// TwinCAT 3 PLC project HMI_Hemo
// ProgramVersion: 3.1.4024.0
// libraries:
//   Tc2_Standard, * (Beckhoff Automation GmbH)
//   Tc2_System, * (Beckhoff Automation GmbH)
//   Tc3_Module, * (Beckhoff Automation GmbH)
//   VisuDialogs, * (System)
//   VisuSymbols,3.5.10.0,System
// project tree:
//   / GlobalTextList.TcGTLO, PlcTask.TcTTO, Visualization Manager.TcVMO (not stored), VISU_TASK.TcTTO
//   GVLs/ GVL.TcGVL
//   POUs/ MAIN.TcPOU
//   VISUs/ Main_Screen.TcVIS, Screen_1.TcVIS, Screen_Maintenance.TcVIS, Screen_1_Sub_1.TcVIS, Screen_1_Sub_2.TcVIS, Screen_1_Sub_3.TcVIS, Screen_1_Sub_4.TcVIS, Screen_3.TcVIS, Screen_3_Sub_1.TcVIS, Screen_2_Sub_1.TcVIS, Screen_2.TcVIS, Screen_2_Sub_2.TcVIS, Screen_2_Sub_7.TcVIS, Screen_2_Sub_6.TcVIS, Screen_2_Sub_3.TcVIS, Screen_2_Sub_4.TcVIS, Screen_2_Sub_5.TcVIS, Screen_Prep.TcVIS, Screen_Rinse.TcVIS, Screen_Dialys.TcVIS
// real-time tasks:
//   TASK PlcTask: cycle T#10ms, priority 20, ADS port 350
//   TASK VISU_TASK: cycle T#200000us, priority 30, ADS port 351

CONFIGURATION HMI_Hemo
    RESOURCE PLC ON TwinCAT3
        TASK PlcTask(INTERVAL := T#10ms, PRIORITY := 20);
        TASK VISU_TASK(INTERVAL := T#200000us, PRIORITY := 30);
        PROGRAM MAIN WITH PlcTask : MAIN;
        PROGRAM VisuElems_Visu_Prg WITH VISU_TASK : VisuElems.Visu_Prg;
    END_RESOURCE
END_CONFIGURATION

// ---- GVLs/GVL.TcGVL
{attribute 'qualified_only'}
VAR_GLOBAL
	
	// HMI State ON/OFF
	HMI_State_ON_OFF				: BOOL;
	
	// HMI Variable Global Heading
	HMI_Heading						: ARRAY[0..2] OF INT;
	
	// HMI Variable Prep
	HMI_Prep_Name_Display			: ARRAY[0..7] OF STRING;
	HMI_Prep_Name_Input				: ARRAY[0..3] OF STRING;
	HMI_Prep_Name_IO				: ARRAY[0..3] OF STRING;
	
	HMI_Prep_Display_Var			: ARRAY[0..7] OF INT;
	HMI_Prep_Input_Var				: ARRAY[0..3] OF INT;
	HMI_Prep_IO_Var					: ARRAY[0..3] OF BOOL;
	
	// HMI Variable Rinse
	HMI_Rinse_Name_Display			: ARRAY[0..7] OF STRING;
	HMI_Rinse_Name_Input				: ARRAY[0..3] OF STRING;
	HMI_Rinse_Name_IO				: ARRAY[0..3] OF STRING;
	
	HMI_Rinse_Display_Var			: ARRAY[0..7] OF INT;
	HMI_Rinse_Input_Var				: ARRAY[0..3] OF INT;
	HMI_Rinse_IO_Var				: ARRAY[0..3] OF BOOL;
	
	// HMI Variable Dialys
	HMI_Dialys_Name_Display			: ARRAY[0..7] OF STRING;
	HMI_Dialys_Name_Input			: ARRAY[0..3] OF STRING;
	HMI_Dialys_Name_IO				: ARRAY[0..3] OF STRING;
	
	HMI_Dialys_Display_Var			: ARRAY[0..7] OF INT;
	HMI_Dialys_Input_Var			: ARRAY[0..3] OF INT;
	HMI_Dialys_IO_Var				: ARRAY[0..3] OF BOOL;
	
	// HMI Variable Global Declaration
	
	HMI_Button_Valve				: ARRAY[0..31] OF BOOL;
	HMI_Display_Int					: ARRAY[0..31] OF INT;
	HMI_Display_Lamp				: ARRAY[0..31] OF BOOL;

	HMI_Motor_Peristaltik_Input 	: INT;
	HMI_Motor_Peristaltik_Real		: INT;
	
	HMI_Motor_DAC_1_Input			: INT;
	HMI_Motor_DAC_1_Real			: INT;
	
	HMI_Motor_DAC_2_Input			: INT;
	HMI_Motor_DAC_2_Real			: INT;
	
	HMI_Motor_Pump_1_Input			: INT;
	HMI_Motor_Pump_1_Real			: INT;
	
	HMI_Motor_Pump_2_Input			: INT;
	HMI_Motor_Pump_2_Real			: INT;
	
	HMI_Motor_Pump_3_Input			: INT;
	HMI_Motor_Pump_3_Real			: INT;
	
	HMI_Motor_Stepper_Input			: INT;
	HMI_Motor_Stepper_Real			: INT;
	HMI_Motor_Stepper_Injec_Stat	: BOOL;
	HMI_Motor_Stepper_Zero_Pos		: BOOL;
	
	HMI_Number_Display				: ARRAY[0..31] OF INT;
	
	//HMI Variable for Maintenance
	
	HMI_Maintenance_H				: BOOL;	
	HMI_Maintenance_P1				: BOOL;	
	HMI_Maintenance_P2				: BOOL;	
	HMI_Maintenance_P3				: BOOL;	
	HMI_Maintenance_P4				: BOOL;	
	
	HMI_Maintenance_V1				: BOOL;	
	HMI_Maintenance_V4				: BOOL;	
	HMI_Maintenance_V5A				: BOOL;	
	HMI_Maintenance_V5B				: BOOL;	
	HMI_Maintenance_V6A				: BOOL;	
	HMI_Maintenance_V6B				: BOOL;	
	HMI_Maintenance_V7A				: BOOL;	
	HMI_Maintenance_V7B				: BOOL;	
	HMI_Maintenance_V8A				: BOOL;	
	HMI_Maintenance_V8B				: BOOL;	
	HMI_Maintenance_V9A				: BOOL;	
	HMI_Maintenance_V9B				: BOOL;

	HMI_Maintenance_V10				: BOOL; 
	HMI_Maintenance_V11				: BOOL;
	HMI_Maintenance_V12				: BOOL;
	HMI_Maintenance_V17				: BOOL;
	HMI_Maintenance_V19				: BOOL;
	HMI_Maintenance_V21				: BOOL;
	HMI_Maintenance_V24				: BOOL;
	HMI_Maintenance_V27				: BOOL;
	HMI_Maintenance_V28				: BOOL;
	HMI_Maintenance_V29				: BOOL;
	HMI_Maintenance_V30				: BOOL;
	HMI_Maintenance_V31				: BOOL;
	
	HMI_Maintenance_V33				: BOOL;	
	HMI_Maintenance_V34				: BOOL;
	HMI_Maintenance_V35				: BOOL;
	HMI_Maintenance_V43				: BOOL;
	HMI_Maintenance_V45				: BOOL;
	HMI_Maintenance_V46				: BOOL;
	HMI_Maintenance_V55				: BOOL;
	HMI_Maintenance_V56				: BOOL;
	HMI_Maintenance_V57				: BOOL;
	
	
	
END_VAR

// ---- POUs/MAIN.TcPOU
PROGRAM MAIN
VAR	

END_VAR

// GVL Variable For Prep
GVL.HMI_Prep_Name_Display[0] := 'Test';
GVL.HMI_Prep_Name_Display[1] := 'Test';
GVL.HMI_Prep_Name_Display[2] := 'Test';
GVL.HMI_Prep_Name_Display[3] := 'Test';
GVL.HMI_Prep_Name_Display[4] := 'Test';
GVL.HMI_Prep_Name_Display[5] := 'Test';
GVL.HMI_Prep_Name_Display[6] := 'Test';
GVL.HMI_Prep_Name_Display[7] := 'Test';

GVL.HMI_Prep_Name_Input[0] := 'Test';
GVL.HMI_Prep_Name_Input[1] := 'Test';
GVL.HMI_Prep_Name_Input[2] := 'Test';
GVL.HMI_Prep_Name_Input[3] := 'Test';

GVL.HMI_Prep_Name_IO[0] := 'Test';
GVL.HMI_Prep_Name_IO[1] := 'Test';
GVL.HMI_Prep_Name_IO[2] := 'Test';
GVL.HMI_Prep_Name_IO[3] := 'Test';

END_PROGRAM

// ---- GlobalTextList.TcGTLO
TEXTLIST GlobalTextList
  52 = ' Val 10: %i'
  420 = ' Val 11: %i'
  658 = ' Val 12: %i'
  696 = ' Val 13: %i'
  313 = ' Val 14: %i'
  1050 = ' Val 15: %i'
  862 = ' Val 16: %i'
  715 = ' Val 17: %i'
  463 = ' Val 18: %i'
  761 = ' Val 19: %i'
  366 = ' Val 1: %i'
  822 = ' Val 20: %i'
  648 = ' Val 21: %i'
  318 = ' Val 22: %i'
  1131 = ' Val 23: %i'
  134 = ' Val 24: %i'
  689 = ' Val 25: %i'
  59 = ' Val 26: %i'
  29 = ' Val 27: %i'
  476 = ' Val 28: %i'
  911 = ' Val 29: %i'
  161 = ' Val 2: %i'
  193 = ' Val 30: %i'
  656 = ' Val 31: %i'
  579 = ' Val 32: %i'
  849 = ' Val 3: %i'
  159 = ' Val 4: %i'
  380 = ' Val 5: %i'
  207 = ' Val 6: %i'
  261 = ' Val 7: %i'
  42 = ' Val 8: %i'
  58 = ' Val 9: %i'
  1018 = '%i'
  1046 = '%s'
  1856 = 'Diagram'
  61 = 'DIALYS'
  1024 = 'Dialys Mode'
  1006 = 'Digital Input'
  1260 = 'Display Variable'
  28 = 'dsfads'
  1374 = 'H'
  608 = 'Injection Status'
  112 = 'Input 1'
  162 = 'Input 10'
  462 = 'Input 11'
  577 = 'Input 12'
  944 = 'Input 13'
  742 = 'Input 14'
  680 = 'Input 15'
  475 = 'Input 16'
  273 = 'Input 17'
  127 = 'Input 18'
  208 = 'Input 19'
  816 = 'Input 2'
  306 = 'Input 20'
  515 = 'Input 21'
  972 = 'Input 22'
  70 = 'Input 23'
  242 = 'Input 24'
  779 = 'Input 25'
  714 = 'Input 26'
  84 = 'Input 27'
  53 = 'Input 28'
  228 = 'Input 29'
  471 = 'Input 3'
  343 = 'Input 30'
  745 = 'Input 31'
  808 = 'Input 32'
  566 = 'Input 4'
  775 = 'Input 5'
  874 = 'Input 6'
  599 = 'Input 7'
  359 = 'Input 8'
  440 = 'Input 9'
  1650 = 'Input Output'
  543 = 'Input Variable'
  1242 = 'Kecepatan Real'
  393 = 'Konfigurasi Input Output'
  931 = 'Konfigurasi Motor'
  633 = 'Lamp 1'
  1869 = 'Maintanance'
  1561 = 'Maintenance'
  544 = 'MAINTENANCE'
  45 = 'Mesin Hemodialisis'
  56 = 'Motor'
  131 = 'Motor DAC 1'
  1109 = 'Motor DAC 2'
  194 = 'Motor Peristaltik'
  744 = 'Motor Pump 1'
  1236 = 'Motor Pump 2'
  304 = 'Motor Pump 3'
  1002 = 'Motor Stepper'
  1079 = 'Num Display 1'
  311 = 'Num Display 2'
  1150 = 'Number Display 1'
  1017 = 'Number Display 2'
  1036 = 'off'
  1043 = 'OFF'
  1929 = 'ON/OFF'
  817 = 'P1'
  60 = 'P2'
  815 = 'P2H'
  649 = 'P3'
  930 = 'P4'
  1144 = 'PREP'
  367 = 'Prep Mode'
  1822 = 'Preparation'
  1625 = 'RINSE'
  1635 = 'Rinse Mode'
  982 = 'Setpoint Kecepatan'
  1174 = 'Tombol Valve'
  678 = 'V1'
  1333 = 'V10'
  617 = 'V11'
  1375 = 'V12'
  1051 = 'V17'
  912 = 'V19'
  1674 = 'V21'
  618 = 'V24'
  542 = 'v27'
  4 = 'V27'
  846 = 'V28'
  922 = 'V29'
  1189 = 'V30'
  510 = 'V31'
  1373 = 'V33'
  1492 = 'V34'
  1774 = 'V35'
  1487 = 'V4'
  593 = 'V43'
  49 = 'V45'
  191 = 'v46'
  101 = 'V46'
  1268 = 'V55'
  1183 = 'V56'
  108 = 'V57'
  66 = 'V5A'
  182 = 'V5a'
  1304 = 'V5b'
  436 = 'V6a'
  1520 = 'V6b'
  468 = 'V7a'
  1310 = 'V7b'
  971 = 'V8a'
  759 = 'V8b'
  200 = 'V9a'
  1329 = 'V9b'
  691 = 'Val 10: %i'
  270 = 'Val 11: %i'
  100 = 'Val 12: %i'
  408 = 'Val 13: %i'
  771 = 'Val 14: %i'
  692 = 'Val 15: %i'
  807 = 'Val 16: %i'
  281 = 'Val 17: %i'
  948 = 'Val 18: %i'
  457 = 'Val 19: %i'
  54 = 'Val 1: %i'
  426 = 'Val 20: %i'
  79 = 'Val 21: %i'
  128 = 'Val 22: %i'
  929 = 'Val 23: %i'
  902 = 'Val 24: %i'
  32 = 'Val 25: %i'
  238 = 'Val 26: %i'
  549 = 'Val 27: %i'
  379 = 'Val 28: %i'
  418 = 'Val 29: %i'
  917 = 'Val 2: %i'
  886 = 'Val 30: %i'
  629 = 'Val 31: %i'
  155 = 'Val 32: %i'
  981 = 'Val 3: %i'
  877 = 'Val 4: %i'
  26 = 'Val 5: %i'
  333 = 'Val 6: %i'
  612 = 'Val 7: %i'
  31 = 'Val 8: %i'
  220 = 'Val 9: %i'
  55 = 'Valve 1'
  964 = 'Valve 10'
  3 = 'Valve 11'
  265 = 'Valve 12'
  952 = 'Valve 13'
  357 = 'Valve 14'
  65 = 'Valve 15'
  664 = 'Valve 16'
  121 = 'Valve 17'
  578 = 'Valve 18'
  589 = 'Valve 19'
  391 = 'Valve 2'
  2 = 'Valve 20'
  954 = 'Valve 21'
  107 = 'Valve 22'
  174 = 'Valve 23'
  934 = 'Valve 24'
  67 = 'Valve 25'
  734 = 'Valve 26'
  354 = 'Valve 27'
  968 = 'Valve 28'
  879 = 'Valve 29'
  502 = 'Valve 3'
  137 = 'Valve 30'
  340 = 'Valve 31'
  348 = 'Valve 32'
  733 = 'Valve 4'
  467 = 'Valve 5'
  227 = 'Valve 6'
  22 = 'Valve 7'
  977 = 'Valve 8'
  737 = 'Valve 9'
  465 = 'Variable Input Output'
  1258 = 'Zero Pos Status'
  464 = 'Zero Position Status'
END_TEXTLIST

// ---- VISUs/Main_Screen.TcVIS
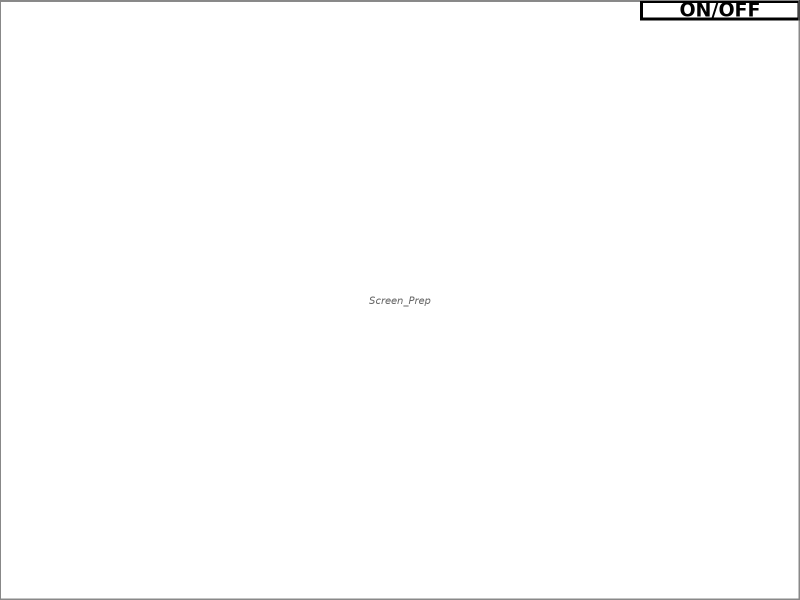
VISUALIZATION Main_Screen  // 800x600
    TabControl (0,1 800x599), frame switch variable: GVL.HMI_Heading[0]
        shows Screen_Prep()
        shows Screen_Rinse()
        shows Screen_Dialys()
        shows Screen_Maintenance()
        [0]: TabTitle=Prep Mode
        [1]: TabTitle=Rinse Mode
        [2]: TabTitle=Dialys Mode
        [3]: TabTitle=Maintenance
    Rectangle (640,0 160x20), "ON/OFF", colour toggle: GVL.HMI_State_ON_OFF
        toggle GVL.HMI_State_ON_OFF
END_VISUALIZATION

// ---- VISUs/Screen_1.TcVIS
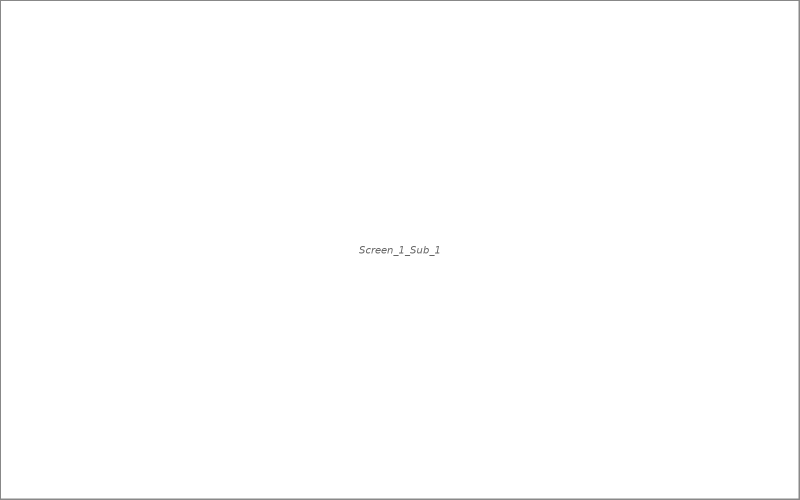
VISUALIZATION Screen_1  // 800x500
    TabControl (0,0 800x500), frame switch variable: GVL.HMI_Heading[2]
        shows Screen_1_Sub_1()
        shows Screen_1_Sub_2()
        shows Screen_1_Sub_3()
        shows Screen_1_Sub_4()
        [0]: TabTitle=Tombol Valve
        [1]: TabTitle=Digital Input
        [2]: TabTitle=Num Display 1
        [3]: TabTitle=Num Display 2
END_VISUALIZATION

// ---- VISUs/Screen_Maintenance.TcVIS
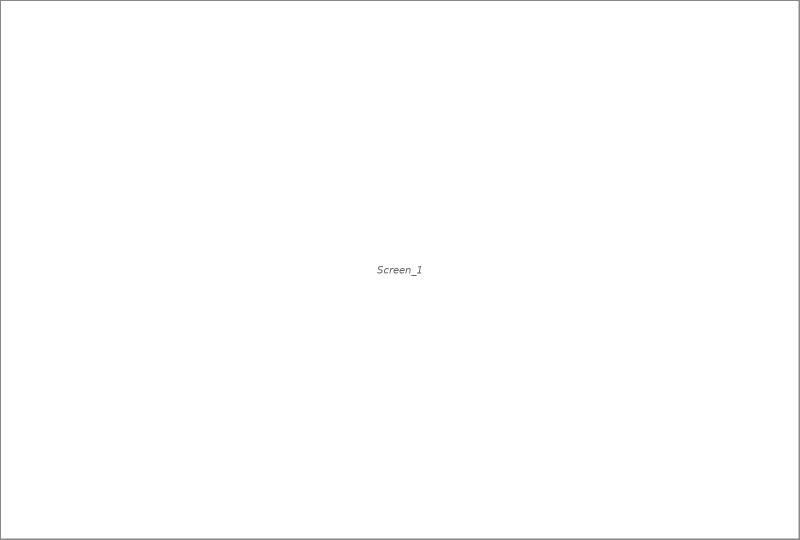
VISUALIZATION Screen_Maintenance  // 800x540
    TabControl (0,0 800x540), frame switch variable: GVL.HMI_Heading[1]
        shows Screen_1()
        shows Screen_2()
        shows Screen_3()
        [0]: TabTitle=Input Output
        [1]: TabTitle=Motor
        [2]: TabTitle=Diagram
END_VISUALIZATION

// ---- VISUs/Screen_1_Sub_1.TcVIS
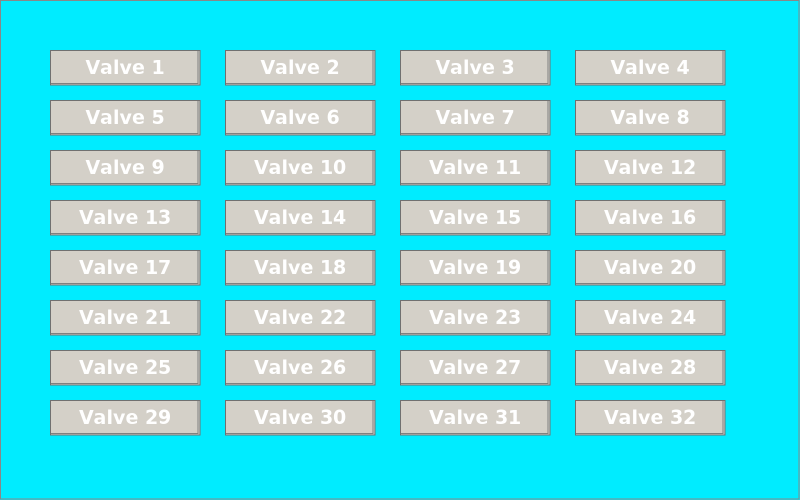
VISUALIZATION Screen_1_Sub_1  // 800x500
    Rectangle (0,0 800x500)
    Button (50,50 150x35), "Valve 1", colour toggle: GVL.HMI_Button_Valve[0]
        toggle GVL.HMI_Button_Valve[0]
    Button (225,50 150x35), "Valve 2", colour toggle: GVL.HMI_Button_Valve[1]
        toggle GVL.HMI_Button_Valve[1] p2164770859=TRUE
    Button (400,50 150x35), "Valve 3", colour toggle: GVL.HMI_Button_Valve[2]
        toggle GVL.HMI_Button_Valve[2] p2164770859=TRUE
    Button (575,50 150x35), "Valve 4", colour toggle: GVL.HMI_Button_Valve[3]
        toggle GVL.HMI_Button_Valve[3] p2164770859=TRUE
    Button (50,100 150x35), "Valve 5", colour toggle: GVL.HMI_Button_Valve[4]
        toggle GVL.HMI_Button_Valve[4] p2164770859=TRUE
    Button (225,100 150x35), "Valve 6", colour toggle: GVL.HMI_Button_Valve[5]
        toggle GVL.HMI_Button_Valve[5] p2164770859=TRUE
    Button (400,100 150x35), "Valve 7", colour toggle: GVL.HMI_Button_Valve[6]
        toggle GVL.HMI_Button_Valve[6] p2164770859=TRUE
    Button (575,100 150x35), "Valve 8", colour toggle: GVL.HMI_Button_Valve[7]
        toggle GVL.HMI_Button_Valve[7] p2164770859=TRUE
    Button (50,150 150x35), "Valve 9", colour toggle: GVL.HMI_Button_Valve[8]
        toggle GVL.HMI_Button_Valve[8] p2164770859=TRUE
    Button (225,150 150x35), "Valve 10", colour toggle: GVL.HMI_Button_Valve[9]
        toggle GVL.HMI_Button_Valve[9] p2164770859=TRUE
    Button (400,150 150x35), "Valve 11", colour toggle: GVL.HMI_Button_Valve[10]
        toggle GVL.HMI_Button_Valve[10] p2164770859=TRUE
    Button (575,150 150x35), "Valve 12", colour toggle: GVL.HMI_Button_Valve[11]
        toggle GVL.HMI_Button_Valve[11] p2164770859=TRUE
    Button (50,200 150x35), "Valve 13", colour toggle: GVL.HMI_Button_Valve[12]
        toggle GVL.HMI_Button_Valve[12] p2164770859=TRUE
    Button (225,200 150x35), "Valve 14", colour toggle: GVL.HMI_Button_Valve[13]
        toggle GVL.HMI_Button_Valve[13] p2164770859=TRUE
    Button (400,200 150x35), "Valve 15", colour toggle: GVL.HMI_Button_Valve[14]
        toggle GVL.HMI_Button_Valve[14] p2164770859=TRUE
    Button (575,200 150x35), "Valve 16", colour toggle: GVL.HMI_Button_Valve[15]
        toggle GVL.HMI_Button_Valve[15] p2164770859=TRUE
    Button (50,250 150x35), "Valve 17", colour toggle: GVL.HMI_Button_Valve[16]
        toggle GVL.HMI_Button_Valve[16] p2164770859=TRUE
    Button (225,250 150x35), "Valve 18", colour toggle: GVL.HMI_Button_Valve[17]
        toggle GVL.HMI_Button_Valve[17] p2164770859=TRUE
    Button (400,250 150x35), "Valve 19", colour toggle: GVL.HMI_Button_Valve[18]
        toggle GVL.HMI_Button_Valve[18] p2164770859=TRUE
    Button (575,250 150x35), "Valve 20", colour toggle: GVL.HMI_Button_Valve[19]
        toggle GVL.HMI_Button_Valve[19] p2164770859=TRUE
    Button (50,300 150x35), "Valve 21", colour toggle: GVL.HMI_Button_Valve[20]
        toggle GVL.HMI_Button_Valve[20] p2164770859=TRUE
    Button (225,300 150x35), "Valve 22", colour toggle: GVL.HMI_Button_Valve[21]
        toggle GVL.HMI_Button_Valve[21] p2164770859=TRUE
    Button (400,300 150x35), "Valve 23", colour toggle: GVL.HMI_Button_Valve[22]
        toggle GVL.HMI_Button_Valve[22] p2164770859=TRUE
    Button (575,300 150x35), "Valve 24", colour toggle: GVL.HMI_Button_Valve[23]
        toggle GVL.HMI_Button_Valve[23] p2164770859=TRUE
    Button (50,350 150x35), "Valve 25", colour toggle: GVL.HMI_Button_Valve[24]
        toggle GVL.HMI_Button_Valve[24] p2164770859=TRUE
    Button (225,350 150x35), "Valve 26", colour toggle: GVL.HMI_Button_Valve[25]
        toggle GVL.HMI_Button_Valve[25] p2164770859=TRUE
    Button (400,350 150x35), "Valve 27", colour toggle: GVL.HMI_Button_Valve[26]
        toggle GVL.HMI_Button_Valve[26] p2164770859=TRUE
    Button (575,350 150x35), "Valve 28", colour toggle: GVL.HMI_Button_Valve[27]
        toggle GVL.HMI_Button_Valve[27] p2164770859=TRUE
    Button (50,400 150x35), "Valve 29", colour toggle: GVL.HMI_Button_Valve[28]
        toggle GVL.HMI_Button_Valve[28] p2164770859=TRUE
    Button (225,400 150x35), "Valve 30", colour toggle: GVL.HMI_Button_Valve[29]
        toggle GVL.HMI_Button_Valve[29] p2164770859=TRUE
    Button (400,400 150x35), "Valve 31", colour toggle: GVL.HMI_Button_Valve[30]
        toggle GVL.HMI_Button_Valve[30] p2164770859=TRUE
    Button (575,400 150x35), "Valve 32", colour toggle: GVL.HMI_Button_Valve[31]
        toggle GVL.HMI_Button_Valve[31] p2164770859=TRUE
END_VISUALIZATION

// ---- VISUs/Screen_1_Sub_2.TcVIS
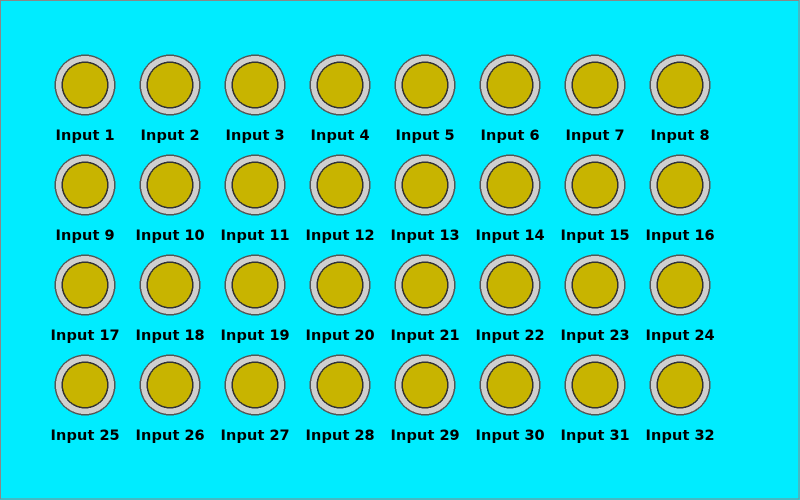
VISUALIZATION Screen_1_Sub_2  // 800x500
    Rectangle (0,0 800x500)
    Lamp1 (50,50 70x70), tooltip "Lamp 1", variable: GVL.HMI_Display_Lamp[0], style: Lamp-Lamp1-Yellow
    Label (50,120 70x30), "Input 1"
    Lamp1 (50,150 70x70), tooltip "Lamp 1", variable: GVL.HMI_Display_Lamp[8], style: Lamp-Lamp1-Yellow
    Label (50,220 70x30), "Input 9"
    Lamp1 (50,250 70x70), tooltip "Lamp 1", variable: GVL.HMI_Display_Lamp[16], style: Lamp-Lamp1-Yellow
    Label (50,320 70x30), "Input 17"
    Lamp1 (50,350 70x70), tooltip "Lamp 1", variable: GVL.HMI_Display_Lamp[24], style: Lamp-Lamp1-Yellow
    Label (50,420 70x30), "Input 25"
    Lamp1 (135,50 70x70), tooltip "Lamp 1", variable: GVL.HMI_Display_Lamp[1], style: Lamp-Lamp1-Yellow
    Label (135,120 70x30), "Input 2"
    Lamp1 (135,150 70x70), tooltip "Lamp 1", variable: GVL.HMI_Display_Lamp[9], style: Lamp-Lamp1-Yellow
    Label (135,220 70x30), "Input 10"
    Lamp1 (135,250 70x70), tooltip "Lamp 1", variable: GVL.HMI_Display_Lamp[17], style: Lamp-Lamp1-Yellow
    Label (135,320 70x30), "Input 18"
    Lamp1 (135,350 70x70), tooltip "Lamp 1", variable: GVL.HMI_Display_Lamp[25], style: Lamp-Lamp1-Yellow
    Label (135,420 70x30), "Input 26"
    Lamp1 (220,50 70x70), tooltip "Lamp 1", variable: GVL.HMI_Display_Lamp[2], style: Lamp-Lamp1-Yellow
    Label (220,120 70x30), "Input 3"
    Lamp1 (220,150 70x70), tooltip "Lamp 1", variable: GVL.HMI_Display_Lamp[10], style: Lamp-Lamp1-Yellow
    Label (220,220 70x30), "Input 11"
    Lamp1 (220,250 70x70), tooltip "Lamp 1", variable: GVL.HMI_Display_Lamp[18], style: Lamp-Lamp1-Yellow
    Label (220,320 70x30), "Input 19"
    Lamp1 (220,350 70x70), tooltip "Lamp 1", variable: GVL.HMI_Display_Lamp[26], style: Lamp-Lamp1-Yellow
    Label (220,420 70x30), "Input 27"
    Lamp1 (305,50 70x70), tooltip "Lamp 1", variable: GVL.HMI_Display_Lamp[3], style: Lamp-Lamp1-Yellow
    Label (305,120 70x30), "Input 4"
    Lamp1 (305,150 70x70), tooltip "Lamp 1", variable: GVL.HMI_Display_Lamp[11], style: Lamp-Lamp1-Yellow
    Label (305,220 70x30), "Input 12"
    Lamp1 (305,250 70x70), tooltip "Lamp 1", variable: GVL.HMI_Display_Lamp[19], style: Lamp-Lamp1-Yellow
    Label (305,320 70x30), "Input 20"
    Lamp1 (305,350 70x70), tooltip "Lamp 1", variable: GVL.HMI_Display_Lamp[27], style: Lamp-Lamp1-Yellow
    Label (305,420 70x30), "Input 28"
    Lamp1 (390,50 70x70), tooltip "Lamp 1", variable: GVL.HMI_Display_Lamp[4], style: Lamp-Lamp1-Yellow
    Label (390,120 70x30), "Input 5"
    Lamp1 (390,150 70x70), tooltip "Lamp 1", variable: GVL.HMI_Display_Lamp[12], style: Lamp-Lamp1-Yellow
    Label (390,220 70x30), "Input 13"
    Lamp1 (390,250 70x70), tooltip "Lamp 1", variable: GVL.HMI_Display_Lamp[20], style: Lamp-Lamp1-Yellow
    Label (390,320 70x30), "Input 21"
    Lamp1 (390,350 70x70), tooltip "Lamp 1", variable: GVL.HMI_Display_Lamp[28], style: Lamp-Lamp1-Yellow
    Label (390,420 70x30), "Input 29"
    Lamp1 (475,50 70x70), tooltip "Lamp 1", variable: GVL.HMI_Display_Lamp[5], style: Lamp-Lamp1-Yellow
    Label (475,120 70x30), "Input 6"
    Lamp1 (475,150 70x70), tooltip "Lamp 1", variable: GVL.HMI_Display_Lamp[13], style: Lamp-Lamp1-Yellow
    Label (475,220 70x30), "Input 14"
    Lamp1 (475,250 70x70), tooltip "Lamp 1", variable: GVL.HMI_Display_Lamp[21], style: Lamp-Lamp1-Yellow
    Label (475,320 70x30), "Input 22"
    Lamp1 (475,350 70x70), tooltip "Lamp 1", variable: GVL.HMI_Display_Lamp[29], style: Lamp-Lamp1-Yellow
    Label (475,420 70x30), "Input 30"
    Lamp1 (560,50 70x70), tooltip "Lamp 1", variable: GVL.HMI_Display_Lamp[6], style: Lamp-Lamp1-Yellow
    Label (560,120 70x30), "Input 7"
    Lamp1 (560,150 70x70), tooltip "Lamp 1", variable: GVL.HMI_Display_Lamp[14], style: Lamp-Lamp1-Yellow
    Label (560,220 70x30), "Input 15"
    Lamp1 (560,250 70x70), tooltip "Lamp 1", variable: GVL.HMI_Display_Lamp[22], style: Lamp-Lamp1-Yellow
    Label (560,320 70x30), "Input 23"
    Lamp1 (560,350 70x70), tooltip "Lamp 1", variable: GVL.HMI_Display_Lamp[30], style: Lamp-Lamp1-Yellow
    Label (560,420 70x30), "Input 31"
    Lamp1 (645,50 70x70), tooltip "Lamp 1", variable: GVL.HMI_Display_Lamp[7], style: Lamp-Lamp1-Yellow
    Label (645,120 70x30), "Input 8"
    Lamp1 (645,150 70x70), tooltip "Lamp 1", variable: GVL.HMI_Display_Lamp[15], style: Lamp-Lamp1-Yellow
    Label (645,220 70x30), "Input 16"
    Lamp1 (645,250 70x70), tooltip "Lamp 1", variable: GVL.HMI_Display_Lamp[23], style: Lamp-Lamp1-Yellow
    Label (645,320 70x30), "Input 24"
    Lamp1 (645,350 70x70), tooltip "Lamp 1", variable: GVL.HMI_Display_Lamp[31], style: Lamp-Lamp1-Yellow
    Label (645,420 70x30), "Input 32"
END_VISUALIZATION

// ---- VISUs/Screen_1_Sub_3.TcVIS
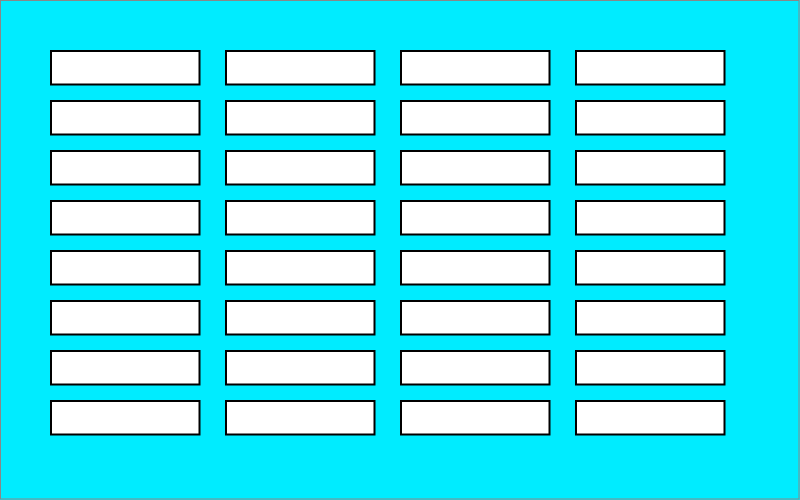
VISUALIZATION Screen_1_Sub_3  // 800x500
    Rectangle (0,0 800x500)
    Rectangle (50,50 150x35), "Val 1: %i", text variable: GVL.HMI_Display_Int[0]
    Rectangle (225,50 150x35), "Val 2: %i", text variable: GVL.HMI_Display_Int[1]
    Rectangle (400,50 150x35), "Val 3: %i", text variable: GVL.HMI_Display_Int[2]
    Rectangle (575,50 150x35), "Val 4: %i", text variable: GVL.HMI_Display_Int[3]
    Rectangle (50,100 150x35), "Val 5: %i", text variable: GVL.HMI_Display_Int[4]
    Rectangle (225,100 150x35), "Val 6: %i", text variable: GVL.HMI_Display_Int[5]
    Rectangle (400,100 150x35), "Val 7: %i", text variable: GVL.HMI_Display_Int[6]
    Rectangle (575,100 150x35), "Val 8: %i", text variable: GVL.HMI_Display_Int[7]
    Rectangle (50,150 150x35), "Val 9: %i", text variable: GVL.HMI_Display_Int[8]
    Rectangle (225,150 150x35), "Val 10: %i", text variable: GVL.HMI_Display_Int[9]
    Rectangle (400,150 150x35), "Val 11: %i", text variable: GVL.HMI_Display_Int[10]
    Rectangle (575,150 150x35), "Val 12: %i", text variable: GVL.HMI_Display_Int[11]
    Rectangle (50,200 150x35), "Val 13: %i", text variable: GVL.HMI_Display_Int[12]
    Rectangle (225,200 150x35), "Val 14: %i", text variable: GVL.HMI_Display_Int[13]
    Rectangle (400,200 150x35), "Val 15: %i", text variable: GVL.HMI_Display_Int[14]
    Rectangle (575,200 150x35), "Val 16: %i", text variable: GVL.HMI_Display_Int[15]
    Rectangle (50,250 150x35), "Val 17: %i", text variable: GVL.HMI_Display_Int[16]
    Rectangle (225,250 150x35), "Val 18: %i", text variable: GVL.HMI_Display_Int[17]
    Rectangle (400,250 150x35), "Val 19: %i", text variable: GVL.HMI_Display_Int[18]
    Rectangle (575,250 150x35), "Val 20: %i", text variable: GVL.HMI_Display_Int[19]
    Rectangle (50,300 150x35), "Val 21: %i", text variable: GVL.HMI_Display_Int[20]
    Rectangle (225,300 150x35), "Val 22: %i", text variable: GVL.HMI_Display_Int[21]
    Rectangle (400,300 150x35), "Val 23: %i", text variable: GVL.HMI_Display_Int[22]
    Rectangle (575,300 150x35), "Val 24: %i", text variable: GVL.HMI_Display_Int[23]
    Rectangle (50,350 150x35), "Val 25: %i", text variable: GVL.HMI_Display_Int[24]
    Rectangle (225,350 150x35), "Val 26: %i", text variable: GVL.HMI_Display_Int[25]
    Rectangle (400,350 150x35), "Val 27: %i", text variable: GVL.HMI_Display_Int[26]
    Rectangle (575,350 150x35), "Val 28: %i", text variable: GVL.HMI_Display_Int[27]
    Rectangle (50,400 150x35), "Val 29: %i", text variable: GVL.HMI_Display_Int[28]
    Rectangle (225,400 150x35), "Val 30: %i", text variable: GVL.HMI_Display_Int[29]
    Rectangle (400,400 150x35), "Val 31: %i", text variable: GVL.HMI_Display_Int[30]
    Rectangle (575,400 150x35), "Val 32: %i", text variable: GVL.HMI_Display_Int[31]
END_VISUALIZATION

// ---- VISUs/Screen_1_Sub_4.TcVIS
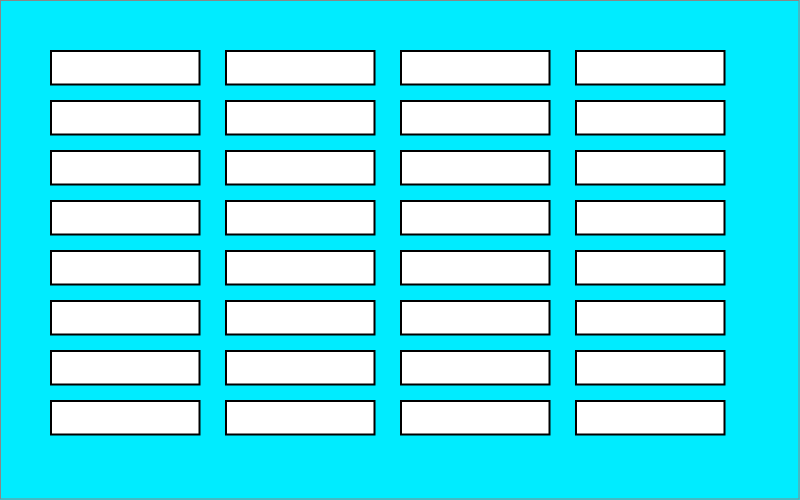
VISUALIZATION Screen_1_Sub_4  // 800x500
    Rectangle (0,0 800x500)
    Rectangle (50,50 150x35), "Val 1: %i", text variable: GVL.HMI_Number_Display[0]
    Rectangle (225,50 150x35), "Val 2: %i", text variable: GVL.HMI_Number_Display[1]
    Rectangle (400,50 150x35), "Val 3: %i", text variable: GVL.HMI_Number_Display[2]
    Rectangle (575,50 150x35), "Val 4: %i", text variable: GVL.HMI_Number_Display[3]
    Rectangle (50,100 150x35), "Val 5: %i", text variable: GVL.HMI_Number_Display[4]
    Rectangle (225,100 150x35), "Val 6: %i", text variable: GVL.HMI_Number_Display[5]
    Rectangle (400,100 150x35), "Val 7: %i", text variable: GVL.HMI_Number_Display[6]
    Rectangle (575,100 150x35), "Val 8: %i", text variable: GVL.HMI_Number_Display[7]
    Rectangle (50,150 150x35), "Val 9: %i", text variable: GVL.HMI_Number_Display[8]
    Rectangle (225,150 150x35), "Val 10: %i", text variable: GVL.HMI_Number_Display[9]
    Rectangle (400,150 150x35), "Val 11: %i", text variable: GVL.HMI_Number_Display[10]
    Rectangle (575,150 150x35), "Val 12: %i", text variable: GVL.HMI_Number_Display[11]
    Rectangle (50,200 150x35), "Val 13: %i", text variable: GVL.HMI_Number_Display[12]
    Rectangle (225,200 150x35), "Val 14: %i", text variable: GVL.HMI_Number_Display[13]
    Rectangle (400,200 150x35), "Val 15: %i", text variable: GVL.HMI_Number_Display[14]
    Rectangle (575,200 150x35), "Val 16: %i", text variable: GVL.HMI_Number_Display[15]
    Rectangle (50,250 150x35), "Val 17: %i", text variable: GVL.HMI_Number_Display[16]
    Rectangle (225,250 150x35), "Val 18: %i", text variable: GVL.HMI_Number_Display[17]
    Rectangle (400,250 150x35), "Val 19: %i", text variable: GVL.HMI_Number_Display[18]
    Rectangle (575,250 150x35), "Val 20: %i", text variable: GVL.HMI_Number_Display[19]
    Rectangle (50,300 150x35), "Val 21: %i", text variable: GVL.HMI_Number_Display[20]
    Rectangle (225,300 150x35), "Val 22: %i", text variable: GVL.HMI_Number_Display[21]
    Rectangle (400,300 150x35), "Val 23: %i", text variable: GVL.HMI_Number_Display[22]
    Rectangle (575,300 150x35), "Val 24: %i", text variable: GVL.HMI_Number_Display[23]
    Rectangle (50,350 150x35), "Val 25: %i", text variable: GVL.HMI_Number_Display[24]
    Rectangle (225,350 150x35), "Val 26: %i", text variable: GVL.HMI_Number_Display[25]
    Rectangle (400,350 150x35), "Val 27: %i", text variable: GVL.HMI_Number_Display[26]
    Rectangle (575,350 150x35), "Val 28: %i", text variable: GVL.HMI_Number_Display[27]
    Rectangle (50,400 150x35), "Val 29: %i", text variable: GVL.HMI_Number_Display[28]
    Rectangle (225,400 150x35), "Val 30: %i", text variable: GVL.HMI_Number_Display[29]
    Rectangle (400,400 150x35), "Val 31: %i", text variable: GVL.HMI_Number_Display[30]
    Rectangle (575,400 150x35), "Val 32: %i", text variable: GVL.HMI_Number_Display[31]
END_VISUALIZATION

// ---- VISUs/Screen_3.TcVIS
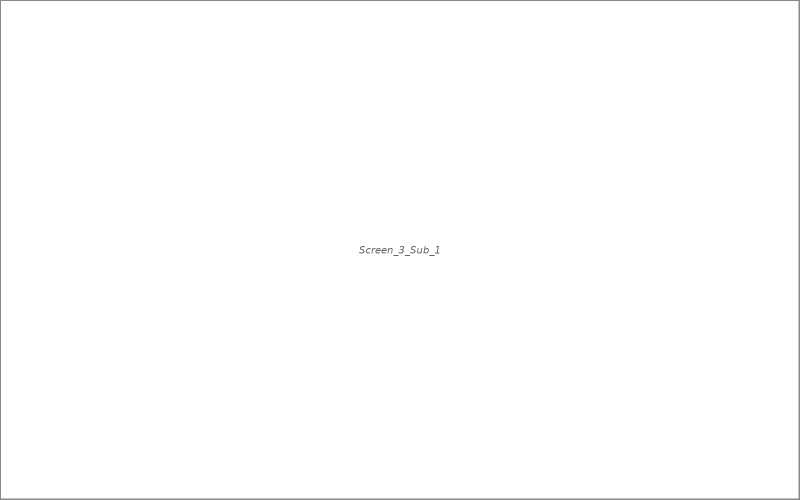
VISUALIZATION Screen_3  // 800x500
    TabControl (0,0 800x500), frame switch variable: GVL.HMI_Heading[2]
        shows Screen_3_Sub_1()
        [0]: TabTitle=Maintenance
END_VISUALIZATION

// ---- VISUs/Screen_3_Sub_1.TcVIS
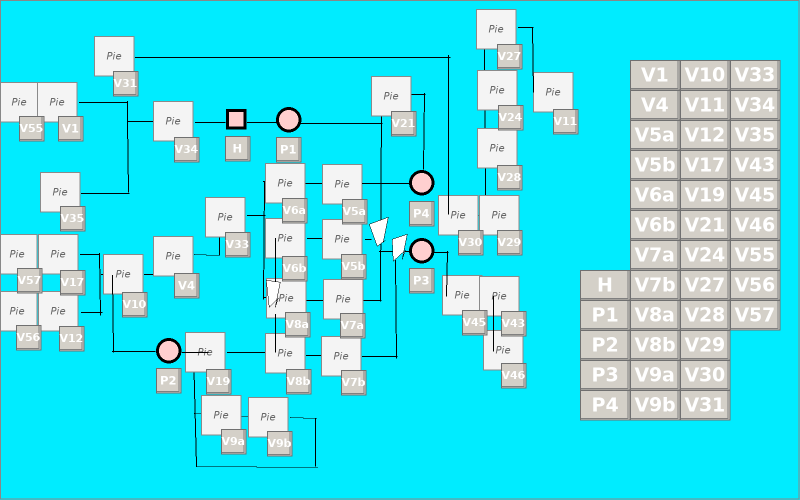
VISUALIZATION Screen_3_Sub_1  // 800x500
    Rectangle (0,0 800x500)
    Line (411,94) (425,94)
    Line (424,93) (423,169)
    Line (380,96) (394,96)
    Line (135,57) (450,57)
    Line (307,238) (342,238)
    Line (42,101) (59,101)
    Line (79,102) (127,102)
    Line (127,121) (175,121)
    Line (81,193) (129,193)
    Line (127,121) (128,192)
    Line (195,122) (225,122)
    Line (247,122) (277,122)
    Line (301,123) (382,123)
    Line (381,96) (380,301)
    Line (380,183) (410,183)
    Line (379,251) (409,251)
    Line (363,300) (381,300)
    Line (306,300) (347,300)
    Line (304,183) (345,183)
    Line (264,181) (263,299)
    Line (263,181) (288,181)
    Line (263,297) (288,297)
    Line (306,355) (341,355)
    Line (275,238) (290,238)
    Line (362,356) (397,356)
    Line (38,254) (59,254)
    Line (39,311) (60,311)
    Line (80,254) (99,254)
    Line (81,312) (102,312)
    Line (101,274) (123,274)
    Line (160,256) (174,255)
    Line (144,274) (162,274)
    Line (160,256) (160,275)
    Line (217,217) (226,217)
    Line (194,254) (218,255)
    Line (219,217) (219,255)
    Line (247,215) (265,215)
    Line (112,351) (155,351)
    Line (227,352) (287,352)
    Line (447,213) (460,214)
    Line (477,215) (503,214)
    Line (484,27) (485,215)
    Line (483,148) (498,148)
    Line (483,89) (498,89)
    Line (483,28) (498,28)
    Line (533,91) (555,91)
    Line (483,295) (501,296)
    Line (433,252) (448,252)
    Line (445,295) (465,295)
    Line (492,350) (505,350)
    Line (193,351) (196,466)
    Line (194,413) (224,414)
    Line (241,416) (271,417)
    Line (290,417) (316,418)
    Line (196,466) (317,467)
    Line (365,239) (371,239)
    Pie (-1,82 40x40), colour toggle: GVL.HMI_Maintenance_V55
    Pie (37,82 40x40), colour toggle: GVL.HMI_Maintenance_V1
    Pie (94,36 40x40), colour toggle: GVL.HMI_Maintenance_V31
    Pie (153,101 40x40), colour toggle: GVL.HMI_Maintenance_V34
    Pie (40,172 40x40), colour toggle: GVL.HMI_Maintenance_V35
    Pie (-3,234 40x40), colour toggle: GVL.HMI_Maintenance_V57
    Pie (-3,291 40x40), colour toggle: GVL.HMI_Maintenance_V56
    Pie (38,234 40x40), colour toggle: GVL.HMI_Maintenance_V17
    Pie (38,291 40x40), colour toggle: GVL.HMI_Maintenance_V12
    Pie (371,76 40x40), colour toggle: GVL.HMI_Maintenance_V21
    Pie (476,9 40x40), colour toggle: GVL.HMI_Maintenance_V27
    Pie (477,70 40x40), colour toggle: GVL.HMI_Maintenance_V24
    Pie (477,128 40x40), colour toggle: GVL.HMI_Maintenance_V28
    Pie (533,72 40x40), colour toggle: GVL.HMI_Maintenance_V11
    Button (580,270 50x30), "H", colour toggle: GVL.HMI_Maintenance_H
        toggle GVL.HMI_Maintenance_H p2164770859=TRUE
    Button (580,300 50x30), "P1", colour toggle: GVL.HMI_Maintenance_P1
        toggle GVL.HMI_Maintenance_P1 p2164770859=TRUE
    Button (580,330 50x30), "P2", colour toggle: GVL.HMI_Maintenance_P2
        toggle GVL.HMI_Maintenance_P2 p2164770859=TRUE
    Button (580,360 50x30), "P3", colour toggle: GVL.HMI_Maintenance_P3
        toggle GVL.HMI_Maintenance_P3 p2164770859=TRUE
    Button (580,390 50x30), "P4", colour toggle: GVL.HMI_Maintenance_P4
        toggle GVL.HMI_Maintenance_P4 p2164770859=TRUE
    Button (630,270 50x30), "V7b", colour toggle: GVL.HMI_Maintenance_V7B
        toggle GVL.HMI_Maintenance_V7B p2164770859=TRUE
    Button (630,300 50x30), "V8a", colour toggle: GVL.HMI_Maintenance_V8A
        toggle GVL.HMI_Maintenance_V8A p2164770859=TRUE
    Button (630,330 50x30), "V8b", colour toggle: GVL.HMI_Maintenance_V8B
        toggle GVL.HMI_Maintenance_V8B p2164770859=TRUE
    Button (630,360 50x30), "V9a", colour toggle: GVL.HMI_Maintenance_V9A
        toggle GVL.HMI_Maintenance_V9A p2164770859=TRUE
    Button (630,390 50x30), "V9b", colour toggle: GVL.HMI_Maintenance_V9B
        toggle GVL.HMI_Maintenance_V9B p2164770859=TRUE
    Button (630,120 50x30), "V5a", colour toggle: GVL.HMI_Maintenance_V5A
        toggle GVL.HMI_Maintenance_V5A p2164770859=TRUE
    Button (630,150 50x30), "V5b", colour toggle: GVL.HMI_Maintenance_V5B
        toggle GVL.HMI_Maintenance_V5B p2164770859=TRUE
    Button (630,180 50x30), "V6a", colour toggle: GVL.HMI_Maintenance_V6A
        toggle GVL.HMI_Maintenance_V6A p2164770859=TRUE
    Button (630,210 50x30), "V6b", colour toggle: GVL.HMI_Maintenance_V6B
        toggle GVL.HMI_Maintenance_V6B p2164770859=TRUE
    Button (630,240 50x30), "V7a", colour toggle: GVL.HMI_Maintenance_V7A
        toggle GVL.HMI_Maintenance_V7A p2164770859=TRUE
    Button (630,60 50x30), "V1", colour toggle: GVL.HMI_Maintenance_V1
        toggle GVL.HMI_Maintenance_V1 p2164770859=TRUE
    Button (630,90 50x30), "V4", colour toggle: GVL.HMI_Maintenance_V4
        toggle GVL.HMI_Maintenance_V4 p2164770859=TRUE
    Button (680,270 50x30), "V27", colour toggle: GVL.HMI_Maintenance_V27
        toggle GVL.HMI_Maintenance_V27 p2164770859=TRUE
    Button (680,300 50x30), "V28", colour toggle: GVL.HMI_Maintenance_V28
        toggle GVL.HMI_Maintenance_V28 p2164770859=TRUE
    Button (680,330 50x30), "V29", colour toggle: GVL.HMI_Maintenance_V29
        toggle GVL.HMI_Maintenance_V29 p2164770859=TRUE
    Button (680,360 50x30), "V30", colour toggle: GVL.HMI_Maintenance_V30
        toggle GVL.HMI_Maintenance_V30 p2164770859=TRUE
    Button (680,390 50x30), "V31", colour toggle: GVL.HMI_Maintenance_V31
        toggle GVL.HMI_Maintenance_V31 p2164770859=TRUE
    Button (680,120 50x30), "V12", colour toggle: GVL.HMI_Maintenance_V12
        toggle GVL.HMI_Maintenance_V12 p2164770859=TRUE
    Button (680,150 50x30), "V17", colour toggle: GVL.HMI_Maintenance_V17
        toggle GVL.HMI_Maintenance_V17 p2164770859=TRUE
    Button (680,180 50x30), "V19", colour toggle: GVL.HMI_Maintenance_V19
        toggle GVL.HMI_Maintenance_V19 p2164770859=TRUE
    Button (680,210 50x30), "V21", colour toggle: GVL.HMI_Maintenance_V21
        toggle GVL.HMI_Maintenance_V21 p2164770859=TRUE
    Button (680,240 50x30), "V24", colour toggle: GVL.HMI_Maintenance_V24
        toggle GVL.HMI_Maintenance_V24 p2164770859=TRUE
    Button (680,60 50x30), "V10", colour toggle: GVL.HMI_Maintenance_V10
        toggle GVL.HMI_Maintenance_V10 p2164770859=TRUE
    Button (680,90 50x30), "V11", colour toggle: GVL.HMI_Maintenance_V11
        toggle GVL.HMI_Maintenance_V11 p2164770859=TRUE
    Button (730,270 50x30), "V56", colour toggle: GVL.HMI_Maintenance_V56
        toggle GVL.HMI_Maintenance_V56 p2164770859=TRUE
    Button (730,300 50x30), "V57", colour toggle: GVL.HMI_Maintenance_V57
        toggle GVL.HMI_Maintenance_V57 p2164770859=TRUE
    Button (730,120 50x30), "V35", colour toggle: GVL.HMI_Maintenance_V35
        toggle GVL.HMI_Maintenance_V35 p2164770859=TRUE
    Button (730,150 50x30), "V43", colour toggle: GVL.HMI_Maintenance_V43
        toggle GVL.HMI_Maintenance_V43 p2164770859=TRUE
    Button (730,180 50x30), "V45", colour toggle: GVL.HMI_Maintenance_V45
        toggle GVL.HMI_Maintenance_V45 p2164770859=TRUE
    Button (730,210 50x30), "V46", colour toggle: GVL.HMI_Maintenance_V46
        toggle GVL.HMI_Maintenance_V46 p2164770859=TRUE
    Button (730,240 50x30), "V55", colour toggle: GVL.HMI_Maintenance_V55
        toggle GVL.HMI_Maintenance_V55 p2164770859=TRUE
    Button (730,60 50x30), "V33", colour toggle: GVL.HMI_Maintenance_V33
        toggle GVL.HMI_Maintenance_V33 p2164770859=TRUE
    Button (730,90 50x30), "V34", colour toggle: GVL.HMI_Maintenance_V34
        toggle GVL.HMI_Maintenance_V34 p2164770859=TRUE
    Button (19,116 25x25), "V55", colour toggle: GVL.HMI_Maintenance_V55
        toggle GVL.HMI_Maintenance_V55 p2164770859=TRUE
    Button (58,116 25x25), "V1", colour toggle: GVL.HMI_Maintenance_V1
        toggle GVL.HMI_Maintenance_V1 p2164770859=TRUE
    Button (113,71 25x25), "V31", colour toggle: GVL.HMI_Maintenance_V31
        toggle GVL.HMI_Maintenance_V31 p2164770859=TRUE
    Button (391,111 25x25), "V21", colour toggle: GVL.HMI_Maintenance_V21
        toggle GVL.HMI_Maintenance_V21 p2164770859=TRUE
    Button (497,44 25x25), "V27", colour toggle: GVL.HMI_Maintenance_V27
        toggle GVL.HMI_Maintenance_V27 p2164770859=TRUE
    Button (498,105 25x25), "V24", colour toggle: GVL.HMI_Maintenance_V24
        toggle GVL.HMI_Maintenance_V24 p2164770859=TRUE
    Button (497,165 25x25), "V28", colour toggle: GVL.HMI_Maintenance_V28
        toggle GVL.HMI_Maintenance_V28 p2164770859=TRUE
    Button (553,109 25x25), "V11", colour toggle: GVL.HMI_Maintenance_V11
        toggle GVL.HMI_Maintenance_V11 p2164770859=TRUE
    Button (174,137 25x25), "V34", colour toggle: GVL.HMI_Maintenance_V34
        toggle GVL.HMI_Maintenance_V34 p2164770859=TRUE
    Button (60,206 25x25), "V35", colour toggle: GVL.HMI_Maintenance_V35
        toggle GVL.HMI_Maintenance_V35 p2164770859=TRUE
    Button (17,268 25x25), "V57", colour toggle: GVL.HMI_Maintenance_V57
        toggle GVL.HMI_Maintenance_V57 p2164770859=TRUE
    Button (60,270 25x25), "V17", colour toggle: GVL.HMI_Maintenance_V17
        toggle GVL.HMI_Maintenance_V17 p2164770859=TRUE
    Button (16,325 25x25), "V56", colour toggle: GVL.HMI_Maintenance_V56
        toggle GVL.HMI_Maintenance_V56 p2164770859=TRUE
    Button (59,326 25x25), "V12", colour toggle: GVL.HMI_Maintenance_V12
        toggle GVL.HMI_Maintenance_V12 p2164770859=TRUE
    Rectangle (226,109 20x20), colour toggle: GVL.HMI_Maintenance_H
    Button (225,136 25x25), "H", colour toggle: GVL.HMI_Maintenance_H
        toggle GVL.HMI_Maintenance_H p2164770859=TRUE
    Ellipse (276,107 25x25), colour toggle: GVL.HMI_Maintenance_P1
    Button (276,137 25x25), "P1", colour toggle: GVL.HMI_Maintenance_P1
        toggle GVL.HMI_Maintenance_P1 p2164770859=TRUE
    Ellipse (156,338 25x25), colour toggle: GVL.HMI_Maintenance_P2
    Button (156,368 25x25), "P2", colour toggle: GVL.HMI_Maintenance_P2
        toggle GVL.HMI_Maintenance_P2 p2164770859=TRUE
    Ellipse (409,238 25x25), colour toggle: GVL.HMI_Maintenance_P3
    Ellipse (409,170 25x25), colour toggle: GVL.HMI_Maintenance_P4
    Button (409,201 25x25), "P4", colour toggle: GVL.HMI_Maintenance_P4
        toggle GVL.HMI_Maintenance_P4 p2164770859=TRUE
    Button (409,268 25x25), "P3", colour toggle: GVL.HMI_Maintenance_P3
        toggle GVL.HMI_Maintenance_P3 p2164770859=TRUE
    Pie (153,236 40x40), colour toggle: GVL.HMI_Maintenance_V4
    Button (174,273 25x25), "V4", colour toggle: GVL.HMI_Maintenance_V4
        toggle GVL.HMI_Maintenance_V4 p2164770859=TRUE
    Pie (103,254 40x40), colour toggle: GVL.HMI_Maintenance_V10
    Button (122,292 25x25), "V10", colour toggle: GVL.HMI_Maintenance_V10
        toggle GVL.HMI_Maintenance_V10 p2164770859=TRUE
    Pie (185,332 40x40), colour toggle: GVL.HMI_Maintenance_V19
    Button (206,369 25x25), "V19", colour toggle: GVL.HMI_Maintenance_V19
        toggle GVL.HMI_Maintenance_V19 p2164770859=TRUE
    Pie (479,195 40x40), colour toggle: GVL.HMI_Maintenance_V29
    Button (497,230 25x25), "V29", colour toggle: GVL.HMI_Maintenance_V29
        toggle GVL.HMI_Maintenance_V29 p2164770859=TRUE
    Pie (438,195 40x40), colour toggle: GVL.HMI_Maintenance_V30
    Button (458,230 25x25), "V30", colour toggle: GVL.HMI_Maintenance_V30
        toggle GVL.HMI_Maintenance_V30 p2164770859=TRUE
    Pie (205,197 40x40), colour toggle: GVL.HMI_Maintenance_V33
    Button (225,232 25x25), "V33", colour toggle: GVL.HMI_Maintenance_V33
        toggle GVL.HMI_Maintenance_V33 p2164770859=TRUE
    Pie (442,275 40x40), colour toggle: GVL.HMI_Maintenance_V45
    Pie (479,276 40x40), colour toggle: GVL.HMI_Maintenance_V43
    Pie (483,330 40x40), colour toggle: GVL.HMI_Maintenance_V46
    Button (462,310 25x25), "V45", colour toggle: GVL.HMI_Maintenance_V45
        toggle GVL.HMI_Maintenance_V45 p2164770859=TRUE
    Button (501,311 25x25), "V43", colour toggle: GVL.HMI_Maintenance_V43
        toggle GVL.HMI_Maintenance_V43 p2164770859=TRUE
    Button (501,363 25x25), "V46", colour toggle: GVL.HMI_Maintenance_V46
        toggle GVL.HMI_Maintenance_V46 p2164770859=TRUE
    Pie (265,163 40x40), colour toggle: GVL.HMI_Maintenance_V6A
    Pie (322,164 40x40), colour toggle: GVL.HMI_Maintenance_V5A
    Pie (265,218 40x40), colour toggle: GVL.HMI_Maintenance_V6B
    Pie (322,219 40x40), colour toggle: GVL.HMI_Maintenance_V5B
    Pie (266,278 40x40), colour toggle: GVL.HMI_Maintenance_V8A
    Pie (323,279 40x40), colour toggle: GVL.HMI_Maintenance_V7A
    Pie (265,333 40x40), colour toggle: GVL.HMI_Maintenance_V8B
    Pie (321,336 40x40), colour toggle: GVL.HMI_Maintenance_V7B
    Button (342,199 25x25), "V5a", colour toggle: GVL.HMI_Maintenance_V5A
        toggle GVL.HMI_Maintenance_V5A p2164770859=TRUE
    Button (341,254 25x25), "V5b", colour toggle: GVL.HMI_Maintenance_V5B
        toggle GVL.HMI_Maintenance_V5B p2164770859=TRUE
    Button (282,198 25x25), "V6a", colour toggle: GVL.HMI_Maintenance_V6A
        toggle GVL.HMI_Maintenance_V6A p2164770859=TRUE
    Button (282,256 25x25), "V6b", colour toggle: GVL.HMI_Maintenance_V6B
        toggle GVL.HMI_Maintenance_V6B p2164770859=TRUE
    Button (340,313 25x25), "V7a", colour toggle: GVL.HMI_Maintenance_V7A
        toggle GVL.HMI_Maintenance_V7A p2164770859=TRUE
    Button (341,370 25x25), "V7b", colour toggle: GVL.HMI_Maintenance_V7B
        toggle GVL.HMI_Maintenance_V7B p2164770859=TRUE
    Button (285,312 25x25), "V8a", colour toggle: GVL.HMI_Maintenance_V8A
        toggle GVL.HMI_Maintenance_V8A p2164770859=TRUE
    Button (286,369 25x25), "V8b", colour toggle: GVL.HMI_Maintenance_V8B
        toggle GVL.HMI_Maintenance_V8B p2164770859=TRUE
    Pie (201,395 40x40), colour toggle: GVL.HMI_Maintenance_V9A
    Pie (248,397 40x40), colour toggle: GVL.HMI_Maintenance_V9B
    Button (221,429 25x25), "V9a", colour toggle: GVL.HMI_Maintenance_V9A
        toggle GVL.HMI_Maintenance_V9A p2164770859=TRUE
    Button (267,431 25x25), "V9b", colour toggle: GVL.HMI_Maintenance_V9B
        toggle GVL.HMI_Maintenance_V9B p2164770859=TRUE
    Line (127,101) (127,121)
    Line (362,183) (384,183)
    Polygon (392,239) (407,234) (402,259) (405,250) (393,261)
    Line (395,260) (396,358)
    Polygon (369,224) (388,217) (383,242) (385,240) (377,246)
    Line (275,238) (275,290)
    Polygon (266,280) (280,282) (275,307) (278,298) (269,307)
    Line (275,314) (275,352)
    Line (99,253) (100,315)
    Line (112,275) (113,352)
    Line (182,352) (208,352)
    Line (448,55) (448,214)
    Line (518,27) (533,27)
    Line (532,27) (533,92)
    Line (447,251) (446,296)
    Line (493,296) (493,351)
    Line (315,418) (315,466)
END_VISUALIZATION

// ---- VISUs/Screen_2_Sub_1.TcVIS
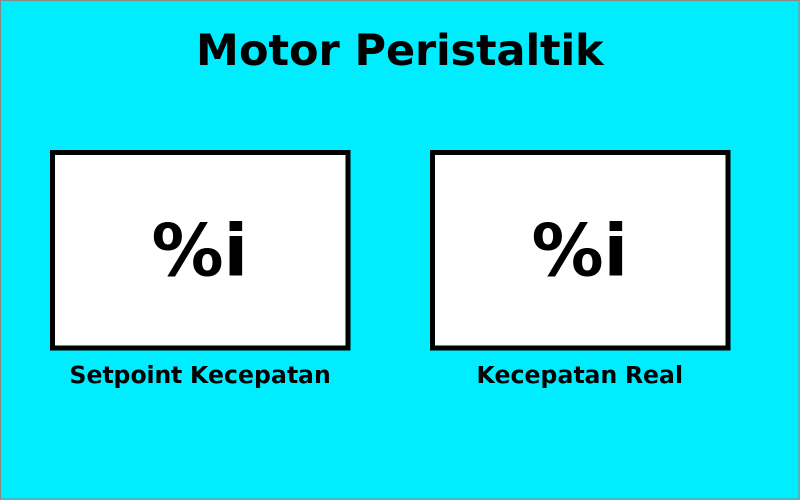
VISUALIZATION Screen_2_Sub_1  // 800x500
    Rectangle (0,0 800x500)
    Label (0,0 800x100), "Motor Peristaltik"
    Rectangle (50,150 300x200), "%i", text variable: GVL.HMI_Motor_Peristaltik_Input
        OnMouseClick: write GVL.HMI_Motor_Peristaltik_Input via VisuDialogs.Numpad
    Label (50,350 300x50), "Setpoint Kecepatan"
    Label (430,350 300x50), "Kecepatan Real"
    Rectangle (430,150 300x200), "%i", text variable: GVL.HMI_Motor_Peristaltik_Real
END_VISUALIZATION

// ---- VISUs/Screen_2.TcVIS
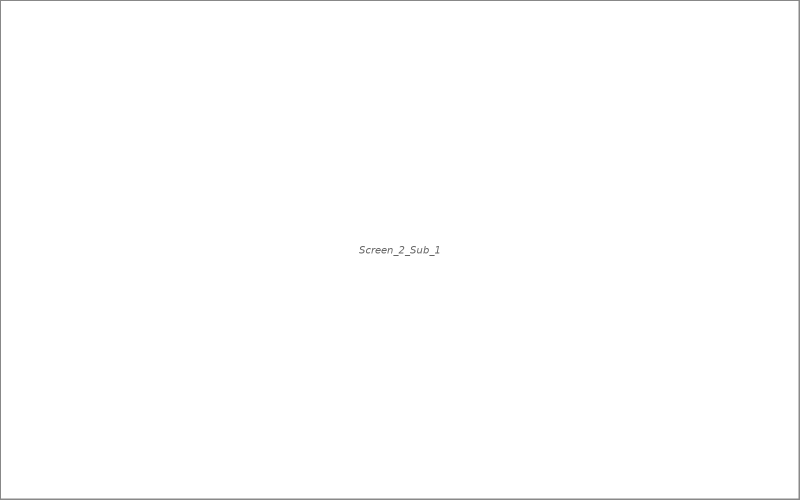
VISUALIZATION Screen_2  // 800x500
    TabControl (0,0 800x500), frame switch variable: GVL.HMI_Heading[2]
        shows Screen_2_Sub_1()
        shows Screen_2_Sub_2()
        shows Screen_2_Sub_6()
        shows Screen_2_Sub_3()
        shows Screen_2_Sub_4()
        shows Screen_2_Sub_7()
        shows Screen_2_Sub_5()
        [0]: TabTitle=Motor Peristaltik
        [1]: TabTitle=Motor DAC 1
        [2]: TabTitle=Motor DAC 2
        [3]: TabTitle=Motor Pump 1
        [4]: TabTitle=Motor Pump 2
        [5]: TabTitle=Motor Pump 3
        [6]: TabTitle=Motor Stepper
END_VISUALIZATION

// ---- VISUs/Screen_2_Sub_2.TcVIS
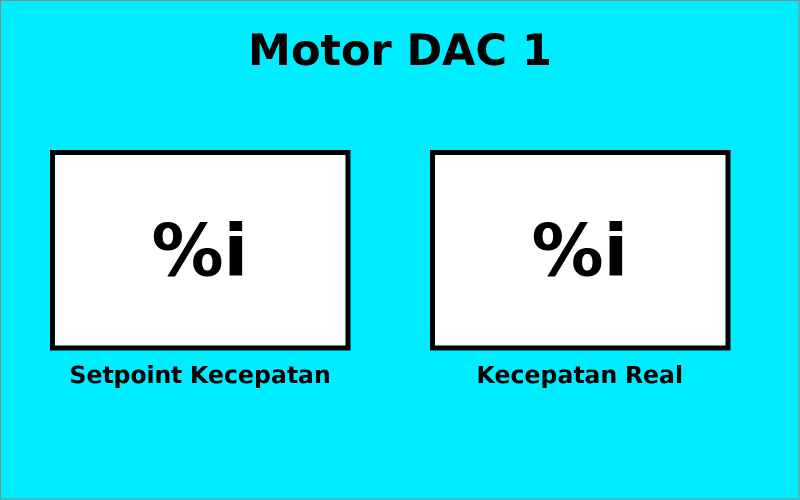
VISUALIZATION Screen_2_Sub_2  // 800x500
    Rectangle (0,0 800x500)
    Label (0,0 800x100), "Motor DAC 1"
    Rectangle (50,150 300x200), "%i", text variable: GVL.HMI_Motor_DAC_1_Input
        OnMouseClick: write GVL.HMI_Motor_DAC_1_Input via VisuDialogs.Numpad
    Label (50,350 300x50), "Setpoint Kecepatan"
    Label (430,350 300x50), "Kecepatan Real"
    Rectangle (430,150 300x200), "%i", text variable: GVL.HMI_Motor_DAC_1_Real
END_VISUALIZATION

// ---- VISUs/Screen_2_Sub_7.TcVIS
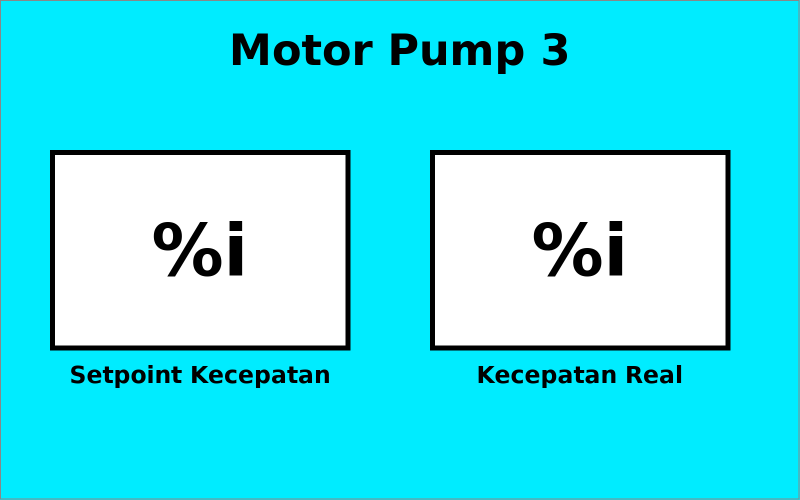
VISUALIZATION Screen_2_Sub_7  // 800x500
    Rectangle (0,0 800x500)
    Label (0,0 800x100), "Motor Pump 3"
    Rectangle (50,150 300x200), "%i", text variable: GVL.HMI_Motor_Pump_3_Input
        OnMouseClick: write GVL.HMI_Motor_Pump_3_Input via VisuDialogs.Numpad
    Label (50,350 300x50), "Setpoint Kecepatan"
    Label (430,350 300x50), "Kecepatan Real"
    Rectangle (430,150 300x200), "%i", text variable: GVL.HMI_Motor_Pump_3_Real
END_VISUALIZATION

// ---- VISUs/Screen_2_Sub_6.TcVIS
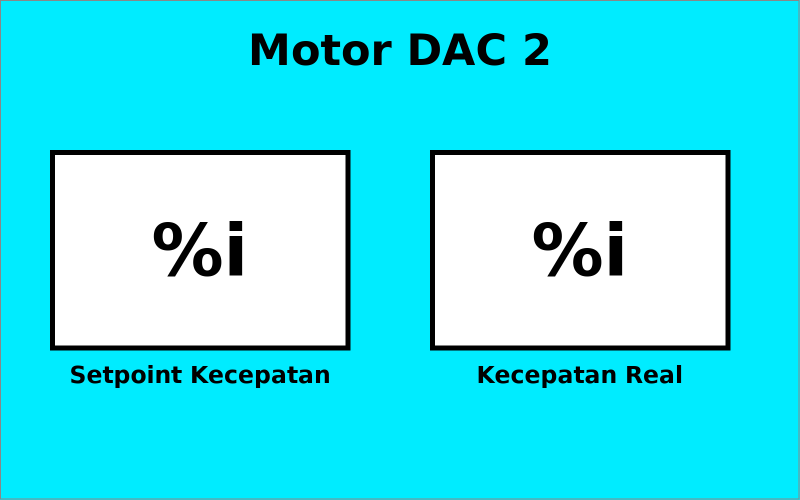
VISUALIZATION Screen_2_Sub_6  // 800x500
    Rectangle (0,0 800x500)
    Label (0,0 800x100), "Motor DAC 2"
    Rectangle (50,150 300x200), "%i", text variable: GVL.HMI_Motor_DAC_2_Input
        OnMouseClick: write GVL.HMI_Motor_DAC_2_Input via VisuDialogs.Numpad
    Label (50,350 300x50), "Setpoint Kecepatan"
    Label (430,350 300x50), "Kecepatan Real"
    Rectangle (430,150 300x200), "%i", text variable: GVL.HMI_Motor_DAC_2_Real
END_VISUALIZATION

// ---- VISUs/Screen_2_Sub_3.TcVIS
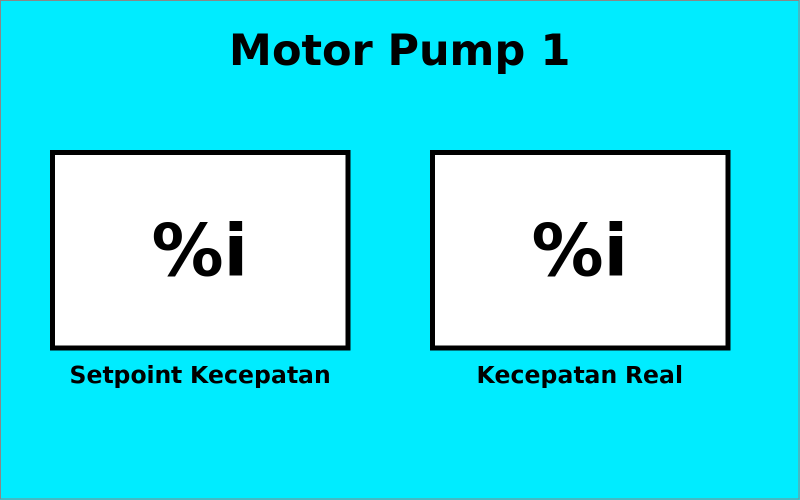
VISUALIZATION Screen_2_Sub_3  // 800x500
    Rectangle (0,0 800x500)
    Label (0,0 800x100), "Motor Pump 1"
    Rectangle (50,150 300x200), "%i", text variable: GVL.HMI_Motor_Pump_1_Input
        OnMouseClick: write GVL.HMI_Motor_Pump_1_Input via VisuDialogs.Numpad
    Label (50,350 300x50), "Setpoint Kecepatan"
    Label (430,350 300x50), "Kecepatan Real"
    Rectangle (430,150 300x200), "%i", text variable: GVL.HMI_Motor_Pump_1_Real
END_VISUALIZATION

// ---- VISUs/Screen_2_Sub_4.TcVIS
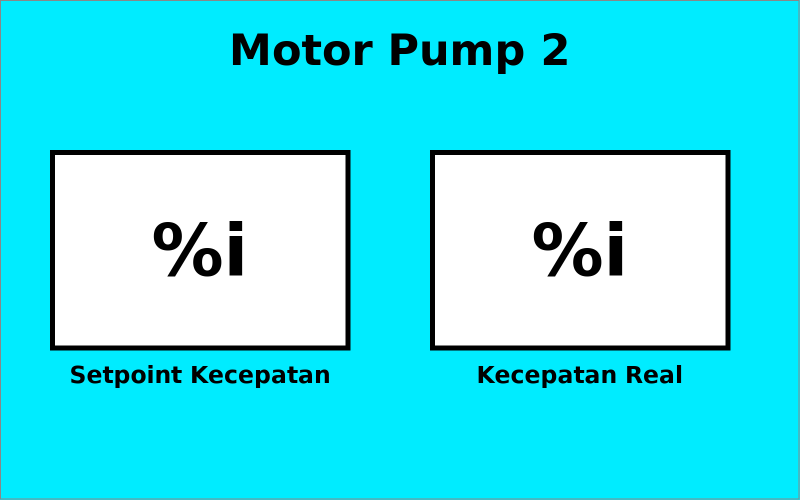
VISUALIZATION Screen_2_Sub_4  // 800x500
    Rectangle (0,0 800x500)
    Label (0,0 800x100), "Motor Pump 2"
    Rectangle (50,150 300x200), "%i", text variable: GVL.HMI_Motor_Pump_2_Input
        OnMouseClick: write GVL.HMI_Motor_Pump_2_Input via VisuDialogs.Numpad
    Label (50,350 300x50), "Setpoint Kecepatan"
    Label (430,350 300x50), "Kecepatan Real"
    Rectangle (430,150 300x200), "%i", text variable: GVL.HMI_Motor_Pump_2_Real
END_VISUALIZATION

// ---- VISUs/Screen_2_Sub_5.TcVIS
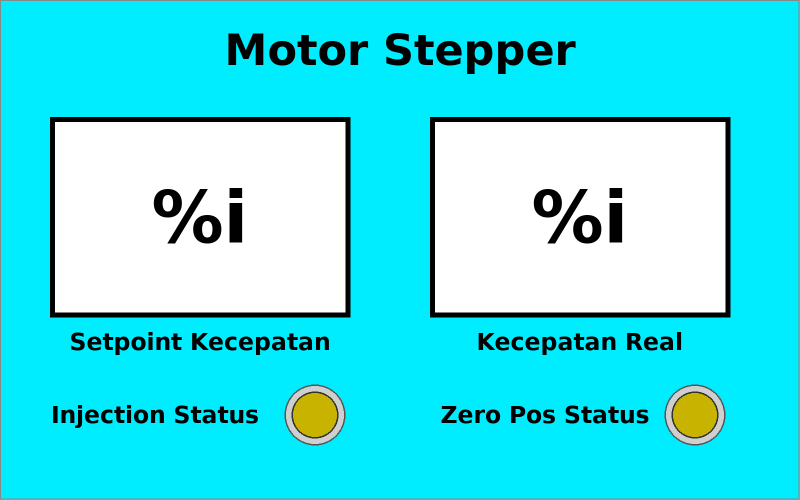
VISUALIZATION Screen_2_Sub_5  // 800x500
    Rectangle (0,0 800x500)
    Label (0,0 800x100), "Motor Stepper"
    Rectangle (50,117 300x200), "%i", text variable: GVL.HMI_Motor_Stepper_Input
        OnMouseClick: write GVL.HMI_Motor_Stepper_Input via VisuDialogs.Numpad
    Label (50,317 300x50), "Setpoint Kecepatan"
    Label (430,317 300x50), "Kecepatan Real"
    Rectangle (430,117 300x200), "%i", text variable: GVL.HMI_Motor_Stepper_Real
    Lamp1 (280,380 70x70), variable: GVL.HMI_Motor_Stepper_Injec_Stat, style: Lamp-Lamp1-Yellow
    Lamp1 (660,380 70x70), variable: GVL.HMI_Motor_Stepper_Zero_Pos, style: Lamp-Lamp1-Yellow
    Label (35,390 240x50), "Injection Status"
    Label (425,390 240x50), "Zero Pos Status"
END_VISUALIZATION

// ---- VISUs/Screen_Prep.TcVIS
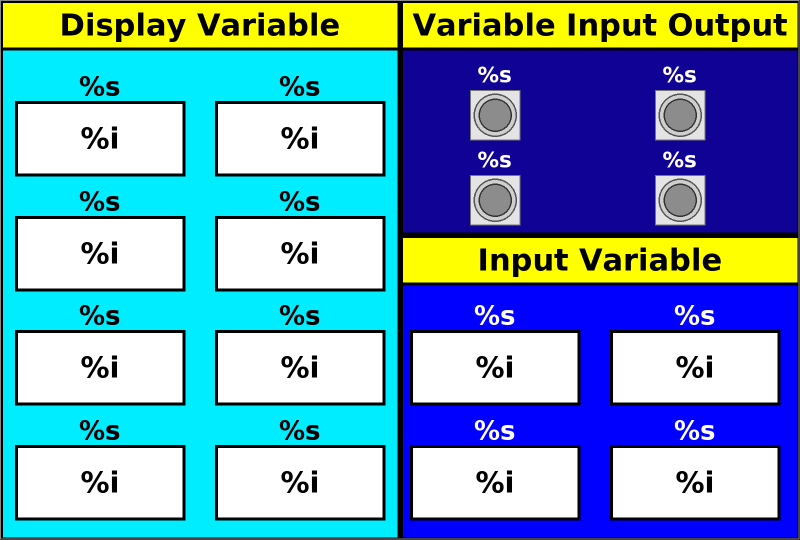
VISUALIZATION Screen_Prep  // 800x540
    Rectangle (400,0 400x235)
    Rectangle (400,235 400x305)
    Rectangle (0,0 400x540)
    Rectangle (15,69 170x35), "%s", text variable: GVL.HMI_Prep_Name_Display[0]
    Rectangle (15,101 170x75), "%i", text variable: GVL.HMI_Prep_Display_Var[0]
    Rectangle (215,69 170x35), "%s", text variable: GVL.HMI_Prep_Name_Display[1]
    Rectangle (215,101 170x75), "%i", text variable: GVL.HMI_Prep_Display_Var[1]
    Rectangle (15,184 170x35), "%s", text variable: GVL.HMI_Prep_Name_Display[2]
    Rectangle (15,216 170x75), "%i", text variable: GVL.HMI_Prep_Display_Var[2]
    Rectangle (215,184 170x35), "%s", text variable: GVL.HMI_Prep_Name_Display[3]
    Rectangle (215,216 170x75), "%i", text variable: GVL.HMI_Prep_Display_Var[3]
    Rectangle (15,298 170x35), "%s", text variable: GVL.HMI_Prep_Name_Display[4]
    Rectangle (15,330 170x75), "%i", text variable: GVL.HMI_Prep_Display_Var[4]
    Rectangle (215,298 170x35), "%s", text variable: GVL.HMI_Prep_Name_Display[5]
    Rectangle (215,330 170x75), "%i", text variable: GVL.HMI_Prep_Display_Var[5]
    Rectangle (15,413 170x35), "%s", text variable: GVL.HMI_Prep_Name_Display[6]
    Rectangle (15,445 170x75), "%i", text variable: GVL.HMI_Prep_Display_Var[6]
    Rectangle (215,413 170x35), "%s", text variable: GVL.HMI_Prep_Name_Display[7]
    Rectangle (215,445 170x75), "%i", text variable: GVL.HMI_Prep_Display_Var[7]
    Rectangle (410,298 170x35), "%s", text variable: GVL.HMI_Prep_Name_Input[0]
    Rectangle (410,330 170x75), "%i", text variable: GVL.HMI_Prep_Input_Var[0]
        OnMouseClick: write GVL.HMI_Prep_Input_Var[0] via VisuDialogs.Numpad
    Rectangle (610,298 170x35), "%s", text variable: GVL.HMI_Prep_Name_Input[1]
    Rectangle (610,330 170x75), "%i", text variable: GVL.HMI_Prep_Input_Var[1]
        OnMouseClick: write GVL.HMI_Prep_Input_Var[1] via VisuDialogs.Numpad
    Rectangle (410,413 170x35), "%s", text variable: GVL.HMI_Prep_Name_Input[2]
    Rectangle (410,445 170x75), "%i", text variable: GVL.HMI_Prep_Input_Var[2]
        OnMouseClick: write GVL.HMI_Prep_Input_Var[2] via VisuDialogs.Numpad
    Rectangle (610,413 170x35), "%s", text variable: GVL.HMI_Prep_Name_Input[3]
    Rectangle (610,445 170x75), "%i", text variable: GVL.HMI_Prep_Input_Var[3]
        OnMouseClick: write GVL.HMI_Prep_Input_Var[3] via VisuDialogs.Numpad
    Rectangle (410,60 170x30), "%s", text variable: GVL.HMI_Prep_Name_IO[0]
    Rectangle (595,60 170x30), "%s", text variable: GVL.HMI_Prep_Name_IO[1]
    Rectangle (410,145 170x30), "%s", text variable: GVL.HMI_Prep_Name_IO[2]
    Rectangle (595,145 170x30), "%s", text variable: GVL.HMI_Prep_Name_IO[3]
    Rectangle (0,0 400x50), "Display Variable"
    Rectangle (400,0 400x50), "Variable Input Output"
    Rectangle (400,235 400x50), "Input Variable"
    PushSwitchLed (470,90 50x50), variable: GVL.HMI_Prep_IO_Var[0], behaviour: TOGGLE, style: Switch-PushSwitchLed-Gray
    PushSwitchLed (655,90 50x50), variable: GVL.HMI_Prep_IO_Var[1], behaviour: TOGGLE, style: Switch-PushSwitchLed-Gray
    PushSwitchLed (655,175 50x50), variable: GVL.HMI_Prep_IO_Var[3], behaviour: TOGGLE, style: Switch-PushSwitchLed-Gray
    PushSwitchLed (470,175 50x50), variable: GVL.HMI_Prep_IO_Var[2], behaviour: TOGGLE, style: Switch-PushSwitchLed-Gray
END_VISUALIZATION

// ---- VISUs/Screen_Rinse.TcVIS
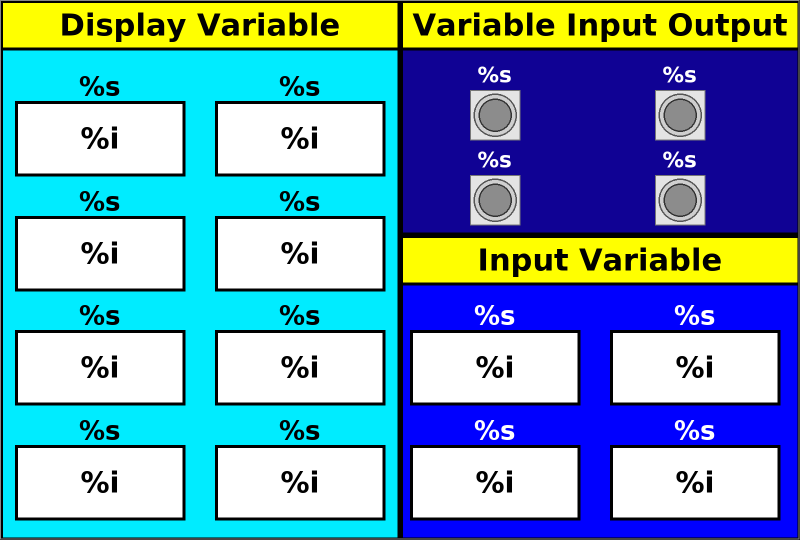
VISUALIZATION Screen_Rinse  // 800x540
    Rectangle (400,0 400x235)
    Rectangle (400,235 400x305)
    Rectangle (0,0 400x540)
    Rectangle (15,69 170x35), "%s", text variable: GVL.HMI_Rinse_Name_Display[0]
    Rectangle (15,101 170x75), "%i", text variable: GVL.HMI_Rinse_Display_Var[0]
    Rectangle (215,69 170x35), "%s", text variable: GVL.HMI_Rinse_Name_Display[1]
    Rectangle (215,101 170x75), "%i", text variable: GVL.HMI_Rinse_Display_Var[1]
    Rectangle (15,184 170x35), "%s", text variable: GVL.HMI_Rinse_Name_Display[2]
    Rectangle (15,216 170x75), "%i", text variable: GVL.HMI_Rinse_Display_Var[2]
    Rectangle (215,184 170x35), "%s", text variable: GVL.HMI_Rinse_Name_Display[3]
    Rectangle (215,216 170x75), "%i", text variable: GVL.HMI_Rinse_Display_Var[3]
    Rectangle (15,298 170x35), "%s", text variable: GVL.HMI_Rinse_Name_Display[4]
    Rectangle (15,330 170x75), "%i", text variable: GVL.HMI_Rinse_Display_Var[4]
    Rectangle (215,298 170x35), "%s", text variable: GVL.HMI_Rinse_Name_Display[5]
    Rectangle (215,330 170x75), "%i", text variable: GVL.HMI_Rinse_Display_Var[5]
    Rectangle (15,413 170x35), "%s", text variable: GVL.HMI_Rinse_Name_Display[6]
    Rectangle (15,445 170x75), "%i", text variable: GVL.HMI_Rinse_Display_Var[6]
    Rectangle (215,413 170x35), "%s", text variable: GVL.HMI_Rinse_Name_Display[7]
    Rectangle (215,445 170x75), "%i", text variable: GVL.HMI_Rinse_Display_Var[7]
    Rectangle (410,298 170x35), "%s", text variable: GVL.HMI_Rinse_Name_Input[0]
    Rectangle (410,330 170x75), "%i", text variable: GVL.HMI_Rinse_Input_Var[0]
        OnMouseClick: write GVL.HMI_Rinse_Input_Var[0] via VisuDialogs.Numpad
    Rectangle (610,298 170x35), "%s", text variable: GVL.HMI_Rinse_Name_Input[1]
    Rectangle (610,330 170x75), "%i", text variable: GVL.HMI_Rinse_Input_Var[1]
        OnMouseClick: write GVL.HMI_Rinse_Input_Var[1] via VisuDialogs.Numpad
    Rectangle (410,413 170x35), "%s", text variable: GVL.HMI_Rinse_Name_Input[2]
    Rectangle (410,445 170x75), "%i", text variable: GVL.HMI_Rinse_Input_Var[2]
        OnMouseClick: write GVL.HMI_Rinse_Input_Var[2] via VisuDialogs.Numpad
    Rectangle (610,413 170x35), "%s", text variable: GVL.HMI_Rinse_Name_Input[3]
    Rectangle (610,445 170x75), "%i", text variable: GVL.HMI_Rinse_Input_Var[3]
        OnMouseClick: write GVL.HMI_Rinse_Input_Var[3] via VisuDialogs.Numpad
    Rectangle (410,60 170x30), "%s", text variable: GVL.HMI_Rinse_Name_IO[0]
    Rectangle (595,60 170x30), "%s", text variable: GVL.HMI_Rinse_Name_IO[1]
    Rectangle (410,145 170x30), "%s", text variable: GVL.HMI_Rinse_Name_IO[2]
    Rectangle (595,145 170x30), "%s", text variable: GVL.HMI_Rinse_Name_IO[3]
    Rectangle (0,0 400x50), "Display Variable"
    Rectangle (400,0 400x50), "Variable Input Output"
    Rectangle (400,235 400x50), "Input Variable"
    PushSwitchLed (470,90 50x50), variable: GVL.HMI_Rinse_IO_Var[0], behaviour: TOGGLE, style: Switch-PushSwitchLed-Gray
    PushSwitchLed (655,90 50x50), variable: GVL.HMI_Rinse_IO_Var[1], behaviour: TOGGLE, style: Switch-PushSwitchLed-Gray
    PushSwitchLed (655,175 50x50), variable: GVL.HMI_Rinse_IO_Var[3], behaviour: TOGGLE, style: Switch-PushSwitchLed-Gray
    PushSwitchLed (470,175 50x50), variable: GVL.HMI_Rinse_IO_Var[2], behaviour: TOGGLE, style: Switch-PushSwitchLed-Gray
END_VISUALIZATION

// ---- VISUs/Screen_Dialys.TcVIS
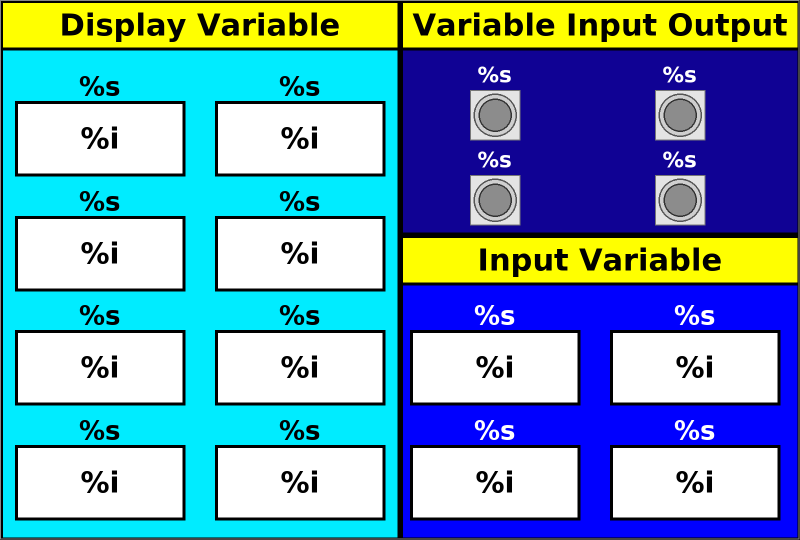
VISUALIZATION Screen_Dialys  // 800x540
    Rectangle (400,0 400x235)
    Rectangle (400,235 400x305)
    Rectangle (0,0 400x540)
    Rectangle (15,69 170x35), "%s", text variable: GVL.HMI_Dialys_Name_Display[0]
    Rectangle (15,101 170x75), "%i", text variable: GVL.HMI_Dialys_Display_Var[0]
    Rectangle (215,69 170x35), "%s", text variable: GVL.HMI_Dialys_Name_Display[1]
    Rectangle (215,101 170x75), "%i", text variable: GVL.HMI_Dialys_Display_Var[1]
    Rectangle (15,184 170x35), "%s", text variable: GVL.HMI_Dialys_Name_Display[2]
    Rectangle (15,216 170x75), "%i", text variable: GVL.HMI_Dialys_Display_Var[2]
    Rectangle (215,184 170x35), "%s", text variable: GVL.HMI_Dialys_Name_Display[3]
    Rectangle (215,216 170x75), "%i", text variable: GVL.HMI_Dialys_Display_Var[3]
    Rectangle (15,298 170x35), "%s", text variable: GVL.HMI_Dialys_Name_Display[4]
    Rectangle (15,330 170x75), "%i", text variable: GVL.HMI_Dialys_Display_Var[4]
    Rectangle (215,298 170x35), "%s", text variable: GVL.HMI_Dialys_Name_Display[5]
    Rectangle (215,330 170x75), "%i", text variable: GVL.HMI_Dialys_Display_Var[5]
    Rectangle (15,413 170x35), "%s", text variable: GVL.HMI_Dialys_Name_Display[6]
    Rectangle (15,445 170x75), "%i", text variable: GVL.HMI_Dialys_Display_Var[6]
    Rectangle (215,413 170x35), "%s", text variable: GVL.HMI_Dialys_Name_Display[7]
    Rectangle (215,445 170x75), "%i", text variable: GVL.HMI_Dialys_Display_Var[7]
    Rectangle (410,298 170x35), "%s", text variable: GVL.HMI_Dialys_Name_Input[0]
    Rectangle (410,330 170x75), "%i", text variable: GVL.HMI_Dialys_Input_Var[0]
        OnMouseClick: write GVL.HMI_Dialys_Input_Var[0] via VisuDialogs.Numpad
    Rectangle (610,298 170x35), "%s", text variable: GVL.HMI_Dialys_Name_Input[1]
    Rectangle (610,330 170x75), "%i", text variable: GVL.HMI_Dialys_Input_Var[1]
        OnMouseClick: write GVL.HMI_Dialys_Input_Var[1] via VisuDialogs.Numpad
    Rectangle (410,413 170x35), "%s", text variable: GVL.HMI_Dialys_Name_Input[2]
    Rectangle (410,445 170x75), "%i", text variable: GVL.HMI_Dialys_Input_Var[2]
        OnMouseClick: write GVL.HMI_Dialys_Input_Var[2] via VisuDialogs.Numpad
    Rectangle (610,413 170x35), "%s", text variable: GVL.HMI_Dialys_Name_Input[3]
    Rectangle (610,445 170x75), "%i", text variable: GVL.HMI_Dialys_Input_Var[3]
        OnMouseClick: write GVL.HMI_Dialys_Input_Var[3] via VisuDialogs.Numpad
    Rectangle (410,60 170x30), "%s", text variable: GVL.HMI_Dialys_Name_IO[0]
    Rectangle (595,60 170x30), "%s", text variable: GVL.HMI_Dialys_Name_IO[1]
    Rectangle (410,145 170x30), "%s", text variable: GVL.HMI_Dialys_Name_IO[2]
    Rectangle (595,145 170x30), "%s", text variable: GVL.HMI_Dialys_Name_IO[3]
    Rectangle (0,0 400x50), "Display Variable"
    Rectangle (400,0 400x50), "Variable Input Output"
    Rectangle (400,235 400x50), "Input Variable"
    PushSwitchLed (470,90 50x50), variable: GVL.HMI_Dialys_IO_Var[0], behaviour: TOGGLE, style: Switch-PushSwitchLed-Gray
    PushSwitchLed (655,90 50x50), variable: GVL.HMI_Dialys_IO_Var[1], behaviour: TOGGLE, style: Switch-PushSwitchLed-Gray
    PushSwitchLed (655,175 50x50), variable: GVL.HMI_Dialys_IO_Var[3], behaviour: TOGGLE, style: Switch-PushSwitchLed-Gray
    PushSwitchLed (470,175 50x50), variable: GVL.HMI_Dialys_IO_Var[2], behaviour: TOGGLE, style: Switch-PushSwitchLed-Gray
END_VISUALIZATION
